PROGRAM MAIN
VAR
END_VAR

PRG_KFE_RIX_VAC_FS();

g_FastFaultOutput2.Execute();

END_PROGRAM

(* stored: Version 1.1.0.1, ProductVersion 3.1.4024.2
   POU MAIN: Id {b903f5d1-e500-41ac-9dbb-336dfebb27d8}, SpecialFunc None *)
